FUNCTION_BLOCK Skill_Greifer_open EXTENDS FB_Skill
VAR_INPUT
	pTool: POINTER TO FB_TOOL;
	Pin: UINT;
	Invert: BOOL := FALSE;
END_VAR
VAR_OUTPUT
END_VAR
VAR
END_VAR

METHOD PROTECTED onActivate : eResult
//set digital output




ADSLOGSTR(ADSLOG_MSGTYPE_HINT, 'Skill Greifer open activated successfull', '');
//check
// if open then
deactivate();


onActivate := eResult.SUCCESS;
END_METHOD

METHOD PROTECTED onCleanup : eResult
onCleanup := eResult.SUCCESS;
END_METHOD

METHOD PROTECTED onConfigure : eResult
onConfigure := eResult.SUCCESS;
END_METHOD

METHOD PROTECTED onDeactivate : eResult
onDeactivate := eResult.SUCCESS;
END_METHOD

METHOD PROTECTED onError : eResult
onError := eResult.SUCCESS;
END_METHOD

METHOD PROTECTED onShutdown : eResult
onShutdown := eResult.SUCCESS;
END_METHOD

END_FUNCTION_BLOCK

(* stored: Version 1.1.0.1, ProductVersion 3.1.4026.18
   POU Skill_Greifer_open: Id {493e94a6-b1d1-445e-8ddf-3f0231b6799c}, SpecialFunc None
   Method onActivate: Id {d7df9868-71f0-4193-acc1-97bc831c4b47}
   Method onCleanup: Id {d4b5b5f4-4752-480e-9c80-7c06e51f9911}
   Method onConfigure: Id {17d6a693-aa18-4118-a60e-1de11ff6cc0e}
   Method onDeactivate: Id {eb63abd5-ca8c-4536-a568-00b2d656c080}
   Method onError: Id {204b9124-02b7-42e8-ad01-ad50412888b7}
   Method onShutdown: Id {0623ac68-704d-43aa-812f-f34b75b26af2} *)
